(* CODESYS project e!C_WagoBeijer_OPCUA_Test_1.ecp

Project tree, tasks and I/O mapping:
  Controller : 750-8202 PFC200 2ETH RS, WAGO, order no. 0750-8202, version 5.11.1.16
    application Application
      libraries: 
      task PLC_Task (cyclic, interval t#10ms, priority 14) calls PLC_PRG
      program PLC_PRG [ST]
      global variables GVL
      Symbols
    DeviceAdapter
    Kbus : Kbus, WAGO, version 1.4.0.2
        unmapped channels: K-BUS diagnostics
    MODBUS
      MODBUS : MODBUS, WAGO, order no. n/a, version 1.1.1.15
    Serial
      COM1 : COM1, WAGO, version 0.0.0.19
*)

// Controller/Application/GVL
{attribute 'qualified_only'}
VAR_GLOBAL
	wGlobalVar1: WORD;
	rGlobalVar2: REAL;
END_VAR

// Controller/Application/PLC_PRG
PROGRAM PLC_PRG
VAR
	rSineAngleTest: REAL;
	wLocalVar1: INT;
END_VAR


PLC_PRG.wLocalVar1 := PLC_PRG.wLocalVar1 + 1;

GVL.wGlobalVar1 := GVL.wGlobalVar1 + 1;

IF (rSineAngleTest < 2*3.14) THEN
	rSineAngleTest := rSineAngleTest + 0.001;
ELSE
	rSineAngleTest := 0;	
END_IF
GVL.rGlobalVar2 := 100 + (100*SIN(rSineAngleTest));

END_PROGRAM
